// Implicitly generated code : DO NOT EDIT
FUNCTION CheckBounds : DINT
VAR_INPUT
	index, lower, upper: DINT;
END_VAR

// Implicitly generated code : Only an Implementation suggestion
{noflow}

Fault_Count_G(CU:=FALSE) ; 
IF  index < lower THEN
	CheckBounds := lower;
	Fault_Count_G(CU:=TRUE) ; 
ELSIF  index > upper THEN
	CheckBounds := upper;
	Fault_Count_G(CU:=TRUE) ; 
ELSE  
	CheckBounds := index;
END_IF
{flow}

END_FUNCTION

(* stored: Version 1.1.0.1, ProductVersion 3.1.4024.2
   POU CheckBounds: Id {9c6aed87-c406-4536-bd74-8348fcf3093f}, SpecialFunc CheckBounds *)
